(* PLC project 20260702.project, Inovance company InoProShop(V1.9.1.6) InoProShop(V1.9.1.6) *)
(* stored: creationDateTime 2026-07-03T21:03:31.881173, modificationDateTime 2026-07-03T19:13:53.8824805 *)

ACTION A11_feed_raise:
            (* FeedLift feed_raise: bounded 1Z jog; final PE1 stable TRUE *)
CASE 上料step OF
	0:
		Z1JOG_pos:=FALSE;
		feedlift_TO(IN:=FALSE, PT:=T#200MS);
		IF FeedLift_1Z_SearchLowTarget >= FeedLift_1Z_SearchHighTarget THEN
			FeedLift_L2_ErrorCode:=303;
			上料step:=0;
			bActionError:=TRUE;
		ELSIF 玻璃上料轴1ZDATE.bHomed AND 玻璃升降接近开关1 AND 上料进料传感器 AND NOT Alarm.0 THEN
			上料step:=10;
		ELSE
			feedlift_TO(IN:=TRUE, PT:=T#10S);
			IF feedlift_TO.Q THEN
				FeedLift_L2_ErrorCode:=301;
				上料step:=0;
				bActionError:=TRUE;
			END_IF
		END_IF
	10:
		feedlift_TO(IN:=FALSE, PT:=T#200MS);
		IF 玻璃升降光电开关1 THEN
			Z1JOG_pos:=FALSE;
			上料step:=20;
		ELSIF 玻璃上料轴1ZDATE.fActPos < FeedLift_1Z_SearchHighTarget THEN
			Z1JOG_pos:=TRUE;
		ELSE
			Z1JOG_pos:=FALSE;
			FeedLift_L2_ErrorCode:=304;
			上料step:=0;
			bActionError:=TRUE;
		END_IF
	20:
		Z1JOG_pos:=FALSE;
		feedlift_TO(IN:=玻璃升降光电开关1, PT:=T#200MS);
		IF feedlift_TO.Q THEN
			上料step:=0;
			bActionDone:=TRUE;
		ELSIF NOT 玻璃升降光电开关1 THEN
			IF 玻璃上料轴1ZDATE.fActPos < FeedLift_1Z_SearchHighTarget THEN
				上料step:=10;
			ELSE
				FeedLift_L2_ErrorCode:=304;
				上料step:=0;
				bActionError:=TRUE;
			END_IF
		END_IF
END_CASE
          
END_ACTION

ACTION A22_unload_bury:
            (* FeedLift unload_bury: bounded 2Z jog to make PE2 stable FALSE; reverse once if low misses *)
CASE 下料step OF
	0:
		Z2JOG_POS:=FALSE;
		Z2JOG_NEG:=FALSE;
		feedlift_TO(IN:=FALSE, PT:=T#200MS);
		IF FeedLift_2Z_SearchLowTarget >= FeedLift_2Z_SearchHighTarget THEN
			FeedLift_L2_ErrorCode:=303;
			下料step:=0;
			bActionError:=TRUE;
		ELSIF 玻璃升降光电开关2 AND 玻璃升降接近开关2 THEN
			下料step:=10;
		ELSE
			feedlift_TO(IN:=TRUE, PT:=T#10S);
			IF feedlift_TO.Q THEN
				FeedLift_L2_ErrorCode:=302;
				下料step:=0;
				bActionError:=TRUE;
			END_IF
		END_IF
	10:
		Z2JOG_POS:=FALSE;
		IF NOT 玻璃升降光电开关2 THEN
			Z2JOG_NEG:=FALSE;
			下料step:=30;
		ELSIF 玻璃上料轴2ZDATE.fActPos > FeedLift_2Z_SearchLowTarget THEN
			Z2JOG_NEG:=TRUE;
		ELSE
			Z2JOG_NEG:=FALSE;
			下料step:=20;
		END_IF
	20:
		Z2JOG_NEG:=FALSE;
		IF NOT 玻璃升降光电开关2 THEN
			Z2JOG_POS:=FALSE;
			下料step:=30;
		ELSIF 玻璃上料轴2ZDATE.fActPos < FeedLift_2Z_SearchHighTarget THEN
			Z2JOG_POS:=TRUE;
		ELSE
			Z2JOG_POS:=FALSE;
			FeedLift_L2_ErrorCode:=305;
			下料step:=0;
			bActionError:=TRUE;
		END_IF
	30:
		Z2JOG_POS:=FALSE;
		Z2JOG_NEG:=FALSE;
		feedlift_TO(IN:=NOT 玻璃升降光电开关2, PT:=T#200MS);
		IF feedlift_TO.Q THEN
			下料step:=0;
			bActionDone:=TRUE;
		ELSIF 玻璃升降光电开关2 THEN
			IF 玻璃上料轴2ZDATE.fActPos > FeedLift_2Z_SearchLowTarget THEN
				下料step:=10;
			ELSIF 玻璃上料轴2ZDATE.fActPos < FeedLift_2Z_SearchHighTarget THEN
				下料step:=20;
			ELSE
				FeedLift_L2_ErrorCode:=305;
				下料step:=0;
				bActionError:=TRUE;
			END_IF
		END_IF
END_CASE
          
END_ACTION

ACTION A91_endcheck:
            (* DEBUG: no-jog photoelectric stable-state confirmation *)
FeedLift_L2_Step := 91;
CASE FeedLift_DebugAxis OF
	1:
		feedlift_TO(IN:=(玻璃升降光电开关1 = FeedLift_DebugExpectedFinal), PT:=T#200MS);
		IF feedlift_TO.Q THEN bActionDone:=TRUE; END_IF
	2:
		feedlift_TO(IN:=(玻璃升降光电开关2 = FeedLift_DebugExpectedFinal), PT:=T#200MS);
		IF feedlift_TO.Q THEN bActionDone:=TRUE; END_IF
ELSE
	FeedLift_L2_ErrorCode:=306;
	bActionError:=TRUE;
END_CASE
          
END_ACTION

ACTION A12_feed_lower:
            (* 上料: 机器人吸住玻璃后, Z1 相对下降 5mm 让位 *)
CASE 上料step OF
	0:
		玻璃上料轴1ZDATE.fRelTarget:=-5.0;
		玻璃上料轴1ZDATE.xMoveRel:=TRUE;
		上料step:=10;
	10:
		IF 玻璃上料轴1ZDATE.bReMoveDone THEN
			玻璃上料轴1ZDATE.xMoveRel:=FALSE;
			上料step:=0;
			bActionDone:=TRUE;
		END_IF
END_CASE

          
END_ACTION

ACTION A21_unload_ready:
            (* FeedLift unload_ready: bounded 2Z search PE2 then leave until PE2 stable FALSE *)
CASE 下料step OF
	0:
		Z2JOG_POS:=FALSE;
		Z2JOG_NEG:=FALSE;
		feedlift_TO(IN:=FALSE, PT:=T#200MS);
		IF FeedLift_2Z_SearchLowTarget >= FeedLift_2Z_SearchHighTarget THEN
			FeedLift_L2_ErrorCode:=303;
			下料step:=0;
			bActionError:=TRUE;
		ELSIF 玻璃上料轴2ZDATE.bHomed AND 下料出料传感器 AND NOT Alarm.1 THEN
			IF 玻璃升降光电开关2 THEN
				下料step:=20;
			ELSE
				下料step:=10;
			END_IF
		ELSE
			feedlift_TO(IN:=TRUE, PT:=T#10S);
			IF feedlift_TO.Q THEN
				FeedLift_L2_ErrorCode:=302;
				下料step:=0;
				bActionError:=TRUE;
			END_IF
		END_IF
	10:
		feedlift_TO(IN:=FALSE, PT:=T#200MS);
		Z2JOG_NEG:=FALSE;
		IF 玻璃升降光电开关2 THEN
			Z2JOG_POS:=FALSE;
			下料step:=20;
		ELSIF 玻璃上料轴2ZDATE.fActPos < FeedLift_2Z_SearchHighTarget THEN
			Z2JOG_POS:=TRUE;
		ELSE
			Z2JOG_POS:=FALSE;
			FeedLift_L2_ErrorCode:=305;
			下料step:=0;
			bActionError:=TRUE;
		END_IF
	20:
		Z2JOG_POS:=FALSE;
		IF NOT 玻璃升降光电开关2 THEN
			Z2JOG_NEG:=FALSE;
			下料step:=30;
		ELSIF 玻璃上料轴2ZDATE.fActPos > FeedLift_2Z_SearchLowTarget THEN
			Z2JOG_NEG:=TRUE;
		ELSE
			Z2JOG_NEG:=FALSE;
			FeedLift_L2_ErrorCode:=305;
			下料step:=0;
			bActionError:=TRUE;
		END_IF
	30:
		Z2JOG_POS:=FALSE;
		Z2JOG_NEG:=FALSE;
		feedlift_TO(IN:=NOT 玻璃升降光电开关2, PT:=T#200MS);
		IF feedlift_TO.Q THEN
			下料step:=0;
			bActionDone:=TRUE;
		ELSIF 玻璃升降光电开关2 THEN
			IF 玻璃上料轴2ZDATE.fActPos > FeedLift_2Z_SearchLowTarget THEN
				下料step:=20;
			ELSE
				FeedLift_L2_ErrorCode:=305;
				下料step:=0;
				bActionError:=TRUE;
			END_IF
		END_IF
END_CASE
          
END_ACTION

PROGRAM FeedLift_L2
  VAR
    上料step : INT;
    下料step : INT;
    bActionDone : BOOL;
    bActionError : BOOL;
    L2_StartTrig : R_TRIG;
    feedlift_TO : TON;
  END_VAR

            (* FeedLift 工位 L2 统一动作派发器
   按 FeedLift_L2_ActionCode 派发到纯设备原子动作 (不含机器人/相机/CNC 握手).
   Start 上升沿接受请求 -> RUNNING 每周期调用对应原子 -> bActionDone=DONE / bActionError=ERROR. *)
L2_StartTrig(CLK := FeedLift_L2_Start);

CASE FeedLift_L2_State OF
	0:  (* IDLE *)
		FeedLift_L2_Step := 0;
		IF L2_StartTrig.Q THEN
			FeedLift_L2_AcceptedSeq := FeedLift_L2_RequestSeq;
			FeedLift_L2_ActiveCode  := FeedLift_L2_ActionCode;
			FeedLift_L2_ErrorCode   := 0;
			FeedLift_L2_Retryable   := FALSE;
			bActionDone  := FALSE;
			bActionError := FALSE;
			上料step := 0;
			下料step := 0;
			CASE FeedLift_L2_ActionCode OF
				11, 12, 21, 22, 91:
					FeedLift_L2_SafeState := 0;
					FeedLift_L2_State     := 10;   (* RUNNING *)
			ELSE
				FeedLift_L2_ErrorCode    := 101;  (* 未知动作码 *)
				FeedLift_L2_Retryable    := TRUE;
				FeedLift_L2_CompletedSeq := FeedLift_L2_AcceptedSeq;
				FeedLift_L2_State        := 30;   (* REJECTED *)
			END_CASE
		END_IF

	10: (* RUNNING *)
		IF FeedLift_L2_Reset THEN FeedLift_L2_State := 0; RETURN; END_IF   (* RUNNING 中 RESET: 中止挂死动作 *)
		CASE FeedLift_L2_ActiveCode OF
			11: A11_feed_raise();
			12: A12_feed_lower();
			21: A21_unload_ready();
			22: A22_unload_bury();
			91: A91_endcheck();
		END_CASE
		IF bActionDone THEN
			bActionDone              := FALSE;
			FeedLift_L2_CompletedSeq := FeedLift_L2_AcceptedSeq;
			FeedLift_L2_State        := 20;   (* DONE *)
		ELSIF bActionError THEN              (* 设备预条件未满足 -> 报错交上位机 *)
			bActionError             := FALSE;
			FeedLift_L2_Retryable    := TRUE;
			FeedLift_L2_CompletedSeq := FeedLift_L2_AcceptedSeq;
			FeedLift_L2_State        := 40;   (* ERROR; ErrorCode 由原子置 *)
		END_IF

	20, 30, 40, 50:  (* 终态: 等 Start 落沿或 Reset 回 IDLE *)
		IF (NOT FeedLift_L2_Start) OR FeedLift_L2_Reset THEN
			FeedLift_L2_State := 0;
		END_IF
END_CASE
          
END_PROGRAM
